(* IEC 61131-3 sources: CodesysTest/alpha/export/FBs/Components, 2 files *)

(* ---- FB_BaggerHeadRaise.pou.st ---- *)
(*#-#-#-#-#-#-#-#-#-#---Declaration---#-#-#-#-#-#-#-#-#-#-#-#-#*)

FUNCTION_BLOCK FB_BaggerHeadRaise
VAR_INPUT
	raiseCommand : BOOL;
	lowerCommand : BOOL;
	raiseLimitSwitch : BOOL;
	lowerLimitSwitch : BOOL;
END_VAR
VAR_OUTPUT
	runMotorOutput : BOOL;
	motorDirectionOutput : BOOL;
END_VAR
VAR
END_VAR
(*#-#-#-#-#-#-#-#-#-#---Implementation---#-#-#-#-#-#-#-#-#-#-#-#-#*)

IF (raiseCommand AND NOT raiseLimitSwitch) OR (lowerCommand AND NOT lowerLimitSwitch) THEN
	runMotorOutput := TRUE;
ELSE
	runMotorOutput := FALSE;
END_IF

IF (lowerCommand AND NOT lowerLimitSwitch) THEN
	motorDirectionOutput := TRUE;
ELSE
	motorDirectionOutput := FALSE;
END_IF

(* ---- HeadRaiseLowerFB.pou.st ---- *)
(*#-#-#-#-#-#-#-#-#-#---Declaration---#-#-#-#-#-#-#-#-#-#-#-#-#*)

FUNCTION_BLOCK HeadRaiseLowerFB
VAR_INPUT
	upperLimitProx : BOOL;
	lowerLimitProx : BOOL;
	raiseCommand : BOOL;
	lowerCommand : BOOL;
END_VAR
VAR_OUTPUT
	raiseOutput : BOOL;
	lowerOutput : BOOL;
END_VAR
VAR
END_VAR
(*#-#-#-#-#-#-#-#-#-#---Implementation---#-#-#-#-#-#-#-#-#-#-#-#-#*)

IF raiseCommand AND NOT upperLimitProx THEN
	raiseOutput := TRUE;
ELSE
	raiseOutput := FALSE;
END_IF

IF lowerCommand AND NOT lowerLimitProx THEN
	lowerOutput := TRUE;
ELSE
	lowerOutput := FALSE;
END_IF
